// TIA Portal V18 export
VAR_GLOBAL   // PLC tag table "INGRESSI"
   In_1 AT %I1.0 : Bool;
   In_2 AT %I1.1 : Bool;
   In_3 AT %I1.2 : Bool;
   In_4 AT %I1.3 : Bool;
   In_5 AT %I1.4 : Bool;
   In_6 AT %I1.5 : Bool;
   In AT %IB1 : Byte;
END_VAR
